PROGRAM MAIN
VAR
	bEnable : BOOL;
	bStart: BOOL;
	nINT: INT:= -32768;
	nUINT: UINT:= 65535;
	fREAL: REAL:= 255.255;
	sPowerStatus : STRING:= 'Power Off';
	nFloatConversion: INT:= 3;
	fFloatConversion: REAL;
	nIntConv: INT;
	fFloatConv: REAL:= 3.3;
END_VAR

bEnable := bStart;

fFloatConversion := INT_TO_REAL(nFloatConversion);
nIntConv := REAL_TO_INT(fFloatConv);

END_PROGRAM

(* stored: Version 1.1.0.1, ProductVersion 3.1.4024.12
   POU MAIN: Id {27431354-f292-4955-aec1-6253c27d76ab}, SpecialFunc None *)
